// Mitsubishi GX Works2 project: 230927-008-A1+A1.A3   PLC: Q03UDV

// task Task_01 (event TRUE, interval 0, priority 31): POU_01

PROGRAM POU_01
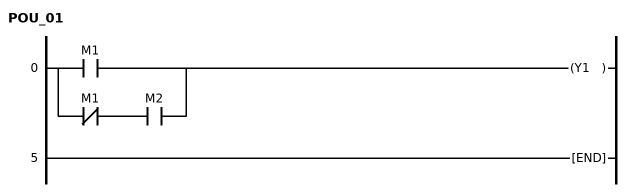
0     LD      M1
      LDI     M1
      AND     M2
      ORB
      OUT     Y1
5     END
END_PROGRAM
